Staubli VAL3: JointState.pjx

--- JointState.pjx ---
Parameters version=s7.7.2 stackSize=5000 millimeterUnit=true
Program file=start.pgx
Program file=stop.pgx
Data file=JointState.dtx

--- JointState.dtx ---
public num nSeq
public num nJoints[10]
